// TwinCAT 3 PLC project Semafor
// ProgramVersion: 3.1.4024.0
// libraries:
//   Tc2_Standard, * (Beckhoff Automation GmbH)
//   Tc2_System, * (Beckhoff Automation GmbH)
//   Tc3_Module, * (Beckhoff Automation GmbH)
//   VisuDialogs, * (System)
// project tree:
//   / GlobalTextList.TcGTLO, PlcTask.TcTTO, Visualization Manager.TcVMO (not stored)
//   POUs/ Blinker.TcPOU, Traffic.TcPOU, MAIN.TcPOU, TrafficLight.TcPOU, Visualization.TcVIS
// real-time tasks:
//   TASK PlcTask: cycle T#10ms, priority 20, ADS port 350

CONFIGURATION Semafor
    RESOURCE PLC ON TwinCAT3
        TASK PlcTask(INTERVAL := T#10ms, PRIORITY := 20);
        PROGRAM MAIN WITH PlcTask : MAIN;
    END_RESOURCE
END_CONFIGURATION

// ---- POUs/MAIN.TcPOU
PROGRAM MAIN
VAR	
END_VAR

TrafficLight(); // calling the function

END_PROGRAM

// ---- POUs/TrafficLight.TcPOU
PROGRAM TrafficLight
VAR
	fbTraffic : Traffic; //declaring the function block in the program
	
	iRedColor : INT;  //integers connected with the hmi that control how much time we input
	iYellowColor : INT;
	iGreenColor : INT; 
	
	bRedLight : BOOL; //bool variables that turn the lights on/off through the hmi
	bYellowLight : BOOL;
	bGreenLight : BOOL;
	
	bTurnOn : BOOL; //bool variable that turns the traffic light on/off
	
	bTempActive : BOOL;	// bool variable that sets/resets the time inserted by the user through hmi
	bTextError : BOOL; //bool variable that makes the textbox for error visible/invisible
END_VAR

fbTraffic.iRedIn := iRedColor; //inputing the time durations in the function block's inputs
fbTraffic.iYellowIn := iYellowColor;
fbTraffic.iGreenIn := iGreenColor;

fbTraffic.bActivate := bTempActive; //activating the input for the time duration status

fbTraffic.bStart := bTurnOn; //inputing the status of the traffic light (on/off)

bTextError := fbTraffic.bError;

bRedLight := fbTraffic.bRed; //the bool variables take the status for the lights and switch them on/off accordingly
bYellowLight := fbTraffic.bYellow;
bGreenLight := fbTraffic.bGreen;

fbTraffic(); // calling the function block

END_PROGRAM

// ---- POUs/Traffic.TcPOU
FUNCTION_BLOCK Traffic
VAR_INPUT	
	bStart : BOOL; //bool variable thats connected with the traffic light status in the program

	iRedIn : INT; //integer variables connected with the time duration integers in the program
	iYellowIn : INT;
	iGreenIn : INT;
	iTimeGreenNew : INT;
	
	bActivate : BOOL;	// bool variable that sets the time duration into the program	
END_VAR
VAR_OUTPUT
	bRed : BOOL;  // bool variables which output the state of the lights (on/off)
	bYellow : BOOL;
	bGreen : BOOL;
	
	bError : BOOL;	 //error bool variables if true makes the error invisible if false makes it visible	
END_VAR
VAR
	fbTimerSt : TON; //timers for every light time duration
	fbTimerRed : TON; 
	fbTimerYR : TON; 
	fbTimerGreen : TON;
	fbTimerYellow : TON; 
	fbTimerReset : TON; 
	fbTimerBlink : TON;
	
	fbBlinker : Blinker; //blinker function block, makes the green light blink
	
	fbTrigger : R_TRIG; //trigger for setting the values (so it doesn't accumuate multiplication)
	
	fbMsgTrigger : R_TRIG; //trigger for a pop up msg
	
	fbMsgTrigger1 : R_TRIG; //trigger for green error output
	
	tTimeRed : TIME; //time variables for the timers
	tTimeYellow : TIME;
	tTimeGreen : TIME;	
END_VAR


IF iRedIn > iYellowIn AND iGreenIn > iYellowIn AND iGreenIn > 3 THEN //checking if yellow's time duration is greater or not than the other time durations
	fbMsgTrigger(CLK := FALSE); //sets the trigger clk to false for the pop up msg
	fbMsgTrigger1(CLK := FALSE); //sets the trigger1 clk to false for the pop up msg
	bError := TRUE; //sets the error to true (invisible)
	fbTrigger(CLK := bActivate); //activates the trigger
	IF fbTrigger.Q THEN
		iTimeGreenNew := (iGreenIn * 1000) - 3000; //substracting the blinking value for green
		tTimeRed := INT_TO_TIME(iRedIn*1000); //converting the integer values to time values
		tTimeYellow := INT_TO_TIME(iYellowIn*1000);
		tTimeGreen := INT_TO_TIME(iTimeGreenNew);
	END_IF
	
	IF bStart THEN // we check whether the traffic light is on/off
	
		fbTimerSt.IN := TRUE; //the starting timer starts
		
		IF fbTimerSt.Q THEN   //red light is on
			bRed := TRUE;
			fbTimerRed.IN := TRUE; // red light timer is on
			
		END_IF
		
		IF fbTimerRed.Q THEN //yellow is on as well
			bYellow := TRUE;
			fbTimerYR.IN := TRUE; //timer for yellow starts		
		END_IF
		
		IF fbTimerYR.Q THEN //red and yellow are off,green lights
			bRed := FALSE;
			bYellow := FALSE;
			bGreen := TRUE;
			fbTimerGreen.IN := TRUE; //timer for green starts
			fbBlinker.bStartBlinker := TRUE; 
			fbBlinker();		
		END_IF
		
		IF fbTimerGreen.Q THEN
			bGreen := FALSE; //green light blinks for 3.5s
			fbTimerBlink.IN := TRUE;//timer for blinker starts
			bGreen := fbBlinker.bStatus;			
		END_IF
		
		IF fbTimerBlink.Q THEN //yellow light,green is off
			bGreen := FALSE;
			bYellow := TRUE;
			fbTimerYellow.IN := TRUE; //timer for yellow starts	
		END_IF
		
		IF fbTimerYellow.Q THEN	//red lights, yellow is off
			bGreen := FALSE;
			bYellow := FALSE;
			bRed := TRUE;
			fbTimerReset.IN := TRUE; //timer for reset starts	
			fbBlinker.bStartBlinker := FALSE;		
		END_IF
		
		IF fbTimerReset.Q THEN //all the timers reset for the next cicle
			fbTimerSt.IN := FALSE;
			fbTimerRed.IN := FALSE;
			fbTimerYR.IN := FALSE;
			fbTimerGreen.IN := FALSE;
			fbTimerYellow.IN := FALSE;
			fbTimerReset.IN := FALSE; 
			fbTimerBlink.IN := FALSE;
		END_IF
		
	END_IF
	
	IF NOT bStart THEN //traffic light is off (turns all lights off)
		bRed := FALSE;
		bYellow := FALSE;
		bGreen := FALSE;
	END_IF		
	
	fbTimerBlink(PT := T#3000MS); //timer for blinker
	fbTimerSt(PT := T#500MS); //timer for start
	fbTimerRed(PT := tTimeRed); //timer for red
	fbTimerYR(PT := tTimeYellow); //timer for yellow
	fbTimerGreen(PT := tTimeGreen); //timer for green
	fbTimerYellow(PT := tTimeYellow); //timer for yellow 2nd cicle
	fbTimerReset(PT := T#500MS); //timer for reseting
ELSIF iGreenIn <= 3 THEN
	fbMsgTrigger1(CLK := TRUE); //error message incase we input lower green value than 3s
	IF fbMsgTrigger1.Q THEN
		ADSLOGSTR(msgCtrlMask := ADSLOG_MSGTYPE_ERROR OR ADSLOG_MSGTYPE_MSGBOX,
				msgFmtStr := 'Please re-enter higher time duration than 3s %s',
				strArg := 'for green!');
	END_IF				
ELSE
	bError := FALSE; //if the inputs are wrong makes the error text box visible
	fbMsgTrigger(CLK := TRUE);
	IF fbMsgTrigger.Q THEN //dispays a pop up msg
		ADSLOGSTR(msgCtrlMask := ADSLOG_MSGTYPE_ERROR OR ADSLOG_MSGTYPE_MSGBOX,
			msgFmtStr := 'Please re-enter the time %s',
			strArg := 'durations!');
	END_IF		
END_IF

END_FUNCTION_BLOCK

// ---- POUs/Blinker.TcPOU
FUNCTION_BLOCK Blinker
VAR_INPUT
	bStartBlinker : BOOL; //bool variable that starts the blinker
END_VAR
VAR_OUTPUT
	bStatus : BOOL; //bool variable that transfers the blinkers output status to the light
END_VAR
VAR
	fbTimer1 : TON; //timers for every on/off state
	fbTimer2 : TON;
	fbTimer3 : TON;
END_VAR

IF bStartBlinker THEN // if the blinker starts execute
	
fbTimer2.IN := TRUE; //starts the time
	IF fbTimer2.Q THEN
		bStatus := FALSE; //sets the light to off
		fbTimer1.IN := TRUE; //starts the new timer
	END_IF

	IF fbTimer1.Q THEN
		bStatus := TRUE; //sets the light to on
		fbTimer3.IN := TRUE; //turns the reset timer
	END_IF
	
	IF fbTimer3.Q THEN
		fbTimer1.IN := FALSE; //resets all the timers
		fbTimer2.IN := FALSE;
		fbTimer3.IN := FALSE;
	END_IF
END_IF
fbTimer1(PT := T#15MS); //timers for the on/off states
fbTimer2(PT := T#15MS);
fbTimer3(PT := T#15MS);

END_FUNCTION_BLOCK

// ---- GlobalTextList.TcGTLO
TEXTLIST GlobalTextList
  977 = '%i Green'
  106 = '%i RED'
  331 = '%i Red'
  226 = '%i Yellow'
  550 = '5000'
  434 = 'Input the time you want each light to last ( in ms)'
  713 = 'Insert the time then click the button to apply changes'
  924 = 'Note: Time is calculated in milliseconds'
  487 = 'OFF'
  911 = 'ON'
  922 = 'Push for ON/OFF'
  196 = 'Set th'
  601 = 'Set the desired time for each light'
  751 = 'Set the desired time for each light '
  801 = 'Set the desired time for each light by clicking'
  799 = 'Set the desired time for each light by clicking on the box'
  381 = 'Start'
  877 = 'Stop'
  540 = 'The inputed value for Yellow is greater'
  575 = 'The inputed value for Yellow is greater than the one for green and red, please '
  362 = 'The inputed value for Yellow is greater than the one for green and red, please reenter values'
  293 = 'TURN OFF'
  462 = 'TURN ON'
END_TEXTLIST

// ---- POUs/Visualization.TcVIS
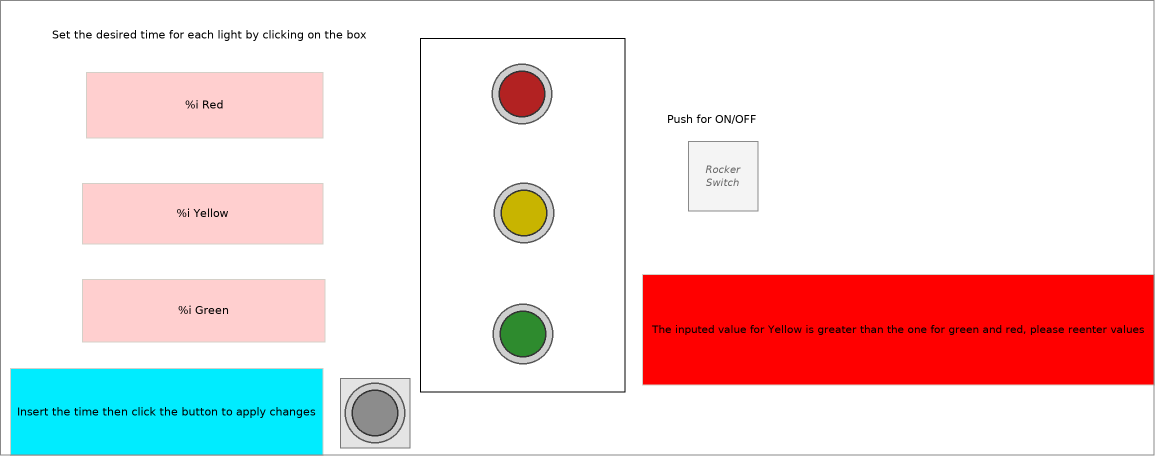
VISUALIZATION Visualization  // 1155x456
    Rectangle (420,38 205x354)
    Lamp1 (487,59 70x70), variable: TrafficLight.bRedLight, style: Lamp-Lamp1-Red
    Lamp1 (489,178 70x70), variable: TrafficLight.bYellowLight, style: Lamp-Lamp1-Yellow
    Lamp1 (488,299 70x70), variable: TrafficLight.bGreenLight, style: Lamp-Lamp1-Green
    Label (34,20 351x30), "Set the desired time for each light by clicking on the box"
    Textfield (86,72 237x66), "%i Red", text variable: TrafficLight.iRedColor
        OnMouseDown: write the text variable via Default
    Textfield (82,183 241x61), "%i Yellow", text variable: TrafficLight.iYellowColor
        OnMouseDown: write the text variable via Default
    Textfield (82,279 243x63), "%i Green", text variable: TrafficLight.iGreenColor
        OnMouseDown: write the text variable via Default
    RockerSwitch (688,141 70x70), variable: TrafficLight.bTurnOn, behaviour: TOGGLE, style: Switch-RockerSwitch-Red
    Label (659,98 106x43), "Push for ON/OFF"
    Textfield (642,274 513x111), "The inputed value for Yellow is greater than the one for green and red, please reenter values", invisible if: TrafficLight.bTextError
    PushSwitch (340,378 70x70), variable: TrafficLight.bTempActive, behaviour: TAP, style: Switch-PushSwitch-Gray
    Textfield (10,368 313x88), "Insert the time then click the button to apply changes"
END_VISUALIZATION
